screen "EQUIPO" 800x480
   GraphicView "Graphic view_1" at 621,5 size 174x31; Picture "LOGO CREMINOX (1)"
   Button "Button_17" at 13,1 size 45x40; TextOff 'Text'; PictureOff "Graphic_3"
      on Click: function_efd93a16()
   TextField "Text field_2" at 71,11 size 93x20; Text 'PARAMETROS'
   Button "Button_30" at 186,4 size 121x32; TextOff 'CONFIGURACION'
      on Click: ActivateScreen("MENU", 0)
   Button "Button_31" at 316,4 size 116x32; TextOff 'CERRAR SESION'
      on Click: function_f23ef4c9()
   Button "Button_12" at 445,5 size 102x32; TextOff 'RECETARIO'
      on Click: ActivateScreen("C RECETAS", 0)
      on Release: ResetBit("HMI RECETARIO")
      on Press: SetBit("HMI RECETARIO")
   TextField "Text field_27" at 301,189 size 50x20; Text 'VAPOR'
      Visibility <- "TIPO DE EQUIPO SELECCIONADO"
   TextField "Text field_28" at 307,208 size 37x20; Text 'VIVO'
      Visibility <- "TIPO DE EQUIPO SELECCIONADO"
   Switch "Switch_2" at 381,188 size 44x40; CaptionText 'Switch'; TextOff 'OFF'; TextOn 'ON'; PictureOn "Graphic_4"; PictureOff "Graphic_5"
      Visibility <- "TIPO DE EQUIPO SELECCIONADO"
      ProcessValue <- "ESTRUCTURAS Y ARREGLOS_HMI CARGA_VAPOR VIVO"
      on SwitchOn: SetBit("ESTRUCTURAS Y ARREGLOS_HMI CARGA_VAPOR VIVO")
      on SwitchOff: ResetBit("ESTRUCTURAS Y ARREGLOS_HMI CARGA_VAPOR VIVO")
   TextField "Text field_6" at 31,96 size 65x22; Text 'T. Agua:'
   IOField "I/O field_3" at 105,96 size 63x24; FormatPattern 99.9; Unit  °C
      ProcessValue <- "ESTRUCTURAS Y ARREGLOS_HMI CARGA_TEMPERATURAS_TEMPERATURA AGUA"
   TextField "Text field_8" at 200,96 size 86x22; Text 'T. Ingreso:'
   IOField "I/O field_4" at 299,96 size 63x24; FormatPattern 99.9; Unit  °C
      ProcessValue <- "ESTRUCTURAS Y ARREGLOS_HMI CARGA_TEMPERATURAS_TEMPERATURA INGRESO"
   TextField "Text field_9" at 391,96 size 63x22; Text 'T. Prod:'
   IOField "I/O field_5" at 468,96 size 63x24; FormatPattern 99.9; Unit  °C
      ProcessValue <- "ESTRUCTURAS Y ARREGLOS_HMI CARGA_TEMPERATURAS_TEMPERATURA PRODUCTO"
   TextField "Text field_7" at 559,96 size 112x22; Text 'Nivel de agua:'
   IOField "I/O field_13" at 686,96 size 69x25; FormatPattern 9999; Unit  mm
      ProcessValue <- "HMI NIVEL"
   TextField "Text field_3" at 28,132 size 153x22; Text 'PRE-OPERACIONAL'
   TextField "Text field_4" at 217,142 size 144x20; Text 'CANTIDAD DE TORRES'
   Button "Button_6" at 386,134 size 36x34; TextOff '-'
      on Press: SetBit("DISMINUIR CANT TORRES")
      on Release: ResetBit("DISMINUIR CANT TORRES")
      Visibility <- "VISUALIZACIONES HMI_LIM INF CANT TORRES"
   IOField "I/O field_6" at 435,133 size 41x35; FormatPattern 99
      ProcessValue <- "ESTRUCTURAS Y ARREGLOS_HMI CARGA_CANTIDAD DE TORRES"
   Button "Button_7" at 490,134 size 36x34; TextOff '+'
      on Press: SetBit("HMI AUMENTAR CANT TORRES")
      on Release: ResetBit("HMI AUMENTAR CANT TORRES")
      Visibility <- "VISUALIZACIONES HMI_LIM SUP CANT TORRES"
   TextField "Text field_23" at 35,210 size 52x20; Text 'TIEMPO'
      Visibility <- "ESTRUCTURAS Y ARREGLOS_HMI CARGA_TIPO DE CORTE"
   IOField "I/O field_1" at 134,202 size 81x32; FormatPattern 999; Unit  min
      ProcessValue <- "ESTRUCTURAS Y ARREGLOS_HMI CARGA_TIEMPO CORTE PC"
      Visibility <- "ESTRUCTURAS Y ARREGLOS_HMI CARGA_TIPO DE CORTE"
   TextField "Text field_5" at 12,178 size 128x20; Text 'POR TEMPERATURA'
   TextField "Text field_10" at 51,160 size 45x20; Text 'CORTE'
   Switch "Switch_1" at 153,159 size 47x38; CaptionText 'Switch'; TextOff 'OFF'; TextOn 'ON'; PictureOn "Graphic_4"; PictureOff "Graphic_5"
      ProcessValue <- "ESTRUCTURAS Y ARREGLOS_HMI CARGA_TIPO DE CORTE"
      on SwitchOn: SetBit("ESTRUCTURAS Y ARREGLOS_HMI CARGA_TIPO DE CORTE")
      on SwitchOff: ResetBit("ESTRUCTURAS Y ARREGLOS_HMI CARGA_TIPO DE CORTE")
   Button "Button_15" at 611,160 size 160x50; TextOff 'INICIAR PRE OP'
      on Release: ResetBit("INICIAR CICLO")
      on Press: SetBit("INICIAR CICLO")
      Visibility <- "ESTRUCTURAS Y ARREGLOS_HMI ESTADO_EN CICLO"
   TextField "Text field_11" at 14,210 size 98x20; Text 'TEMPERATURA'
      Visibility <- "ESTRUCTURAS Y ARREGLOS_HMI CARGA_TIPO DE CORTE"
   IOField "I/O field_15" at 135,202 size 81x32; FormatPattern 999; Unit  °C
      ProcessValue <- "ESTRUCTURAS Y ARREGLOS_HMI CARGA_TEMPERATURA CORTE PC"
      Visibility <- "ESTRUCTURAS Y ARREGLOS_HMI CARGA_TIPO DE CORTE"
   TextField "Text field_12" at 31,243 size 117x22; Text 'OPERACIONAL'
   TextField "Text field_13" at 31,270 size 110x20; Text 'RECETA ELEGIDA'
   TextField "Text field_15" at 31,308 size 129x20; Text 'NOMBRE DE RECETA'
   IOField "I/O field_8" at 196,303 size 221x27; FormatPattern ??????????????????????????
      ProcessValue <- "ESTRUCTURAS Y ARREGLOS_HMI CARGA_NOMBRE RECETA"
   Button "Button_8" at 207,260 size 36x34; TextOff '-'
      on Press: SetBit("HMI SEL ANT RECETA")
      on Release: ResetBit("HMI SEL ANT RECETA")
   IOField "I/O field_7" at 256,260 size 41x35; FormatPattern 99
      ProcessValue <- "HMI RECETA SELECCIONADA"
   Button "Button_9" at 311,261 size 36x34; TextOff '+'
      on Press: SetBit("HMI SEL SIG RECETA")
      on Release: ResetBit("HMI SEL SIG RECETA")
   Button "Button_10" at 367,261 size 129x33; TextOff 'VISUALIZAR'
      on Press: SetBit("HMI VISUALIZAR RECETA")
      on Release: ResetBit("HMI VISUALIZAR RECETA")
      on Click: ActivateScreen("C RECETAS", 0)
   Button "Button_16" at 608,262 size 161x50; TextOff 'INICIAR OPERACIONAL'
      on Release: ResetBit("HMI INICIAR CICLO OP")
      on Press: SetBit("HMI INICIAR CICLO OP")
      Visibility <- "ESTRUCTURAS Y ARREGLOS_HMI ESTADO_EN CICLO"
   TextField "Text field_18" at 30,352 size 114x20; Text 'ESTADO ACTUAL:'
   IOField "I/O field_9" at 153,347 size 251x27; FormatPattern ??????????????????????????????
      ProcessValue <- "ESTRUCTURAS Y ARREGLOS_HMI ESTADO_EQUIPO"
   TextField "Text field_20" at 429,351 size 199x20; Text 'TIEMPO TOTAL TRANSCURRIDO'
      Visibility <- "ESTRUCTURAS Y ARREGLOS_HMI ESTADO_EN CICLO"
   IOField "I/O field_10" at 639,346 size 81x32; FormatPattern 999; Unit  min
      ProcessValue <- "ESTRUCTURAS Y ARREGLOS_HMI ESTADO_TIEMPO TRANSCURRIDO"
      Visibility <- "ESTRUCTURAS Y ARREGLOS_HMI ESTADO_EN CICLO"
   TextField "Text field_21" at 29,392 size 98x20; Text 'PASO ACTUAL'
      Visibility <- "VISUALIZACIONES HMI_PASOS OP EN COCINAS"
   IOField "I/O field_11" at 143,383 size 41x35; FormatPattern 99
      Visibility <- "VISUALIZACIONES HMI_PASOS OP EN COCINAS"
      ProcessValue <- "ESTRUCTURAS Y ARREGLOS_HMI ESTADO_PASO ACTUAL"
   TextField "Text field_22" at 357,393 size 98x20; Text 'TIPO DE CORTE'
      Visibility <- "ESTRUCTURAS Y ARREGLOS_HMI ESTADO_EN CICLO"
   IOField "I/O field_12" at 469,389 size 194x27; FormatPattern ????????????????????
      Visibility <- "ESTRUCTURAS Y ARREGLOS_HMI ESTADO_EN CICLO"
      ProcessValue <- "ESTRUCTURAS Y ARREGLOS_HMI ESTADO_TIPO DE CORTE"
   Rectangle "Rectangle_2" at 1,126 size 798x354
      Visibility <- "ESTRUCTURAS Y ARREGLOS_HMI ESTADO_CICLO FINALIZADO"
   TextField "Text field_14" at 238,145 size 319x43; Text 'CICLO FINALIZADO'
      Visibility <- "ESTRUCTURAS Y ARREGLOS_HMI ESTADO_CICLO FINALIZADO"
   TextField "Text field_17" at 303,198 size 187x43; Text 'CON EXITO'
      Visibility <- "ESTRUCTURAS Y ARREGLOS_HMI ESTADO_CICLO FINALIZADO"
   GraphicView "Graphic view_2" at 348,251 size 98x92; Picture "Graphic_4"
      Visibility <- "ESTRUCTURAS Y ARREGLOS_HMI ESTADO_CICLO FINALIZADO"
   Button "Button_13" at 323,368 size 148x59; TextOff 'OK'
      Visibility <- "ESTRUCTURAS Y ARREGLOS_HMI ESTADO_CICLO FINALIZADO"
      on Press: SetBit("HMI OK FIN DE CICLO")
      on Release: ResetBit("HMI OK FIN DE CICLO")
   Rectangle "Rectangle_3" at 1,126 size 798x354
      Visibility <- "ESTRUCTURAS Y ARREGLOS_HMI ESTADO_CICLO CANCELADO"
   TextField "Text field_19" at 245,166 size 312x43; Text 'CICLO CANCELADO'
      Visibility <- "ESTRUCTURAS Y ARREGLOS_HMI ESTADO_CICLO CANCELADO"
   GraphicView "Graphic view_3" at 357,229 size 86x77; Picture "Graphic_5"
      Visibility <- "ESTRUCTURAS Y ARREGLOS_HMI ESTADO_CICLO CANCELADO"
   Button "Button_14" at 323,331 size 150x61; TextOff 'OK'
      Visibility <- "ESTRUCTURAS Y ARREGLOS_HMI ESTADO_CICLO CANCELADO"
      on Press: SetBit("HMI OK CANCELAR")
      on Release: ResetBit("HMI OK CANCELAR")
   Rectangle "Rectangle_4" at 1,126 size 798x113
      Visibility <- "ESTRUCTURAS Y ARREGLOS_HMI ESTADO_EN PO"
   Rectangle "Rectangle_5" at 1,238 size 798x100
      Visibility <- "ESTRUCTURAS Y ARREGLOS_HMI ESTADO_EN OP"
   Rectangle "Rectangle_6" at 2,128 size 796x112
      Visibility <- "ESTRUCTURAS Y ARREGLOS_HMI ESTADO_EN OP"
   Rectangle "Rectangle_8" at 599,139 size 185x183
      Visibility <- "ESTRUCTURAS Y ARREGLOS_HMI ESTADO_MANUAL ACTIVO"
   TextField "Text field_1" at 609,153 size 154x20; Text 'ACTUADORES ACTIVOS'
      Visibility <- "ESTRUCTURAS Y ARREGLOS_HMI ESTADO_MANUAL ACTIVO"
   TextField "Text field_24" at 623,175 size 127x20; Text 'EN FORMA MANUAL'
      Visibility <- "ESTRUCTURAS Y ARREGLOS_HMI ESTADO_MANUAL ACTIVO"
   Button "Button_11" at 642,261 size 98x38; TextOff 'RESET'
      Visibility <- "ESTRUCTURAS Y ARREGLOS_HMI ESTADO_MANUAL ACTIVO"
      on Press: SetBit("HMI RESET ACTUADORES MANUAL")
      on Release: ResetBit("HMI RESET ACTUADORES MANUAL")
   TextField "Text field_25" at 623,197 size 126x20; Text 'PULSE RESET PARA'
      Visibility <- "ESTRUCTURAS Y ARREGLOS_HMI ESTADO_MANUAL ACTIVO"
   TextField "Text field_26" at 629,220 size 115x20; Text 'DESACTIVARLOS'
      Visibility <- "ESTRUCTURAS Y ARREGLOS_HMI ESTADO_MANUAL ACTIVO"
   Button "Button_3" at 25,429 size 97x43; TextOff 'CANCELAR'
      on Release: ResetBit("HMI CANCELAR")
      on Press: SetBit("HMI CANCELAR")
      Visibility <- "ESTRUCTURAS Y ARREGLOS_HMI ESTADO_PULSADOR CANCELAR"
   Button "Button_4" at 136,430 size 97x43; TextOff 'CONTINUAR'
      on Release: ResetBit("HMI CONTINUAR")
      on Press: SetBit("HMI CONTINUAR")
      Visibility <- "ESTRUCTURAS Y ARREGLOS_HMI ESTADO_PULSADOR CONTINUAR"
   Button "Button_5" at 249,430 size 97x43; TextOff 'PAUSAR'
      on Release: ResetBit("HMI PAUSA")
      on Press: SetBit("HMI PAUSA")
      Visibility <- "ESTRUCTURAS Y ARREGLOS_HMI ESTADO_PULSADOR PAUSA"
   IOField "I/O field_16" at 166,49 size 215x35; FormatPattern ??????????????????????????
      ProcessValue <- "ESTRUCTURAS Y ARREGLOS_HMI NOMBRE EQUIPO"
   Button "Button_19" at 400,49 size 39x35; TextOff 'Text'; PictureOff "Graphic_1"
      on Release: ResetBit("HMI DISMINUIR EQUIPO")
      on Press: SetBit("HMI DISMINUIR EQUIPO")
      Visibility <- "VISUALIZACIONES HMI_LIM INF EQUIPO SEL"
   IOField "I/O field_2" at 464,49 size 42x35; FormatPattern 99
      ProcessValue <- "EQUIPO SELECCIONADO"
   Button "Button_18" at 531,49 size 40x35; TextOff 'Text'; PictureOff "Graphic_2"
      on Release: ResetBit("HMI AUMENTAR EQUIPO")
      on Press: SetBit("HMI AUMENTAR EQUIPO")
      Visibility <- "VISUALIZACIONES HMI_LIM SUP EQUIPO SEL"
   Button "Button_1" at 567,434 size 183x37; TextOff 'GRAFICO TEMPERATURAS'
      on Click: ActivateScreen("GRAFICOS", 0)
   Button "Button_2" at 204,384 size 109x35; TextOff 'SALTAR PASO'
      on Press: SetBit("HMI SALTAR PASO")
      on Release: ResetBit("HMI SALTAR PASO")
      Visibility <- "VISUALIZACIONES HMI_PASOS OP EN COCINAS"

screen "C GENERALES" 800x480
   TextField "Text field_7" at 439,158 size 246x29; Text 'Histeresis temperatura'
   IOField "I/O field_4" at 706,153 size 74x40; FormatPattern 999; Unit  °C
      ProcessValue <- "ESTRUCTURAS Y ARREGLOS_HMI CONFIGURACION_HISTERESIS"
   TextField "Text field_8" at 28,338 size 228x29; Text 'Tiempo Maximo Ciclo'
   IOField "I/O field_5" at 326,333 size 74x40; FormatPattern 999; Unit  min
      ProcessValue <- "ESTRUCTURAS Y ARREGLOS_HMI CONFIGURACION_TIEMPO MAXIMO CICLO"
   IOField "I/O field_3" at 326,242 size 74x40; FormatPattern 9999; Unit  mm
      ProcessValue <- "ESTRUCTURAS Y ARREGLOS_HMI CONFIGURACION_NIVEL CRITICO OP"
   TextField "Text field_9" at 26,158 size 281x29; Text 'Nivel Critico Pre-operativo'
   IOField "I/O field_10" at 326,153 size 74x40; FormatPattern 9999; Unit  mm
      ProcessValue <- "ESTRUCTURAS Y ARREGLOS_HMI CONFIGURACION_NIVEL CRITICO"
   GraphicView "Graphic view_1" at 621,4 size 174x31; Picture "LOGO CREMINOX (1)"
   TextField "Text field_1" at 213,106 size 14x20; Text 'Text'
   Button "Button_1" at 734,430 size 40x35; TextOff 'Text'; PictureOff "Graphic_2"
      on Click: ActivateScreen("C NIVELES PO Y OP", 0)
   Button "Button_4" at 28,430 size 39x35; TextOff 'Text'; PictureOff "Graphic_1"
      on Click: ActivateScreen("C TEMPERATURAS", 0)
   Button "Button_6" at 17,2 size 40x38; TextOff 'Text'; PictureOff "Home"
      on Click: ActivateScreen("PRINCIPAL", 0)
   TextField "Text field_2" at 145,12 size 196x20; Text 'CONFIGURACIONES GENERALES'
   TextField "Text field_3" at 76,439 size 156x18; Text 'A CONF. TEMPERATURAS'
   TextField "Text field_4" at 615,439 size 107x18; Text 'A CONF. NIVELES'
   Button "Button_17" at 83,1 size 45x40; TextOff 'Text'; PictureOff "Graphic_3"
      on Click: ActivateScreen("MENU", 0)
   TextField "Text field_5" at 28,247 size 237x29; Text 'Nivel Critico operativo'
   IOField "I/O field_16" at 166,55 size 215x35; FormatPattern ??????????????????????????
      ProcessValue <- "ESTRUCTURAS Y ARREGLOS_HMI NOMBRE EQUIPO"
   Button "Button_19" at 400,55 size 39x35; TextOff 'Text'; PictureOff "Graphic_1"
      on Release: ResetBit("HMI DISMINUIR EQUIPO")
      on Press: SetBit("HMI DISMINUIR EQUIPO")
      Visibility <- "VISUALIZACIONES HMI_LIM INF EQUIPO SEL"
   IOField "I/O field_1" at 464,55 size 42x35; FormatPattern 99
      ProcessValue <- "EQUIPO SELECCIONADO"
   Button "Button_18" at 531,55 size 40x35; TextOff 'Text'; PictureOff "Graphic_2"
      on Release: ResetBit("HMI AUMENTAR EQUIPO")
      on Press: SetBit("HMI AUMENTAR EQUIPO")
      Visibility <- "VISUALIZACIONES HMI_LIM SUP EQUIPO SEL"

screen "C RECETAS" 800x480
   TextField "Text field_18" at 328,196 size 142x20; Text 'TEMPERATURA CORTE'
      Visibility <- "VISUALIZACIONES HMI_TIPO DE CORTE PASO 1"
   IOField "I/O field_9" at 495,193 size 73x27; FormatPattern 999; Unit  °C
      ProcessValue <- "ESTRUCTURAS Y ARREGLOS_HMI EDICION RECETAS_TEMP PRODUCTO{1}"
      Visibility <- "VISUALIZACIONES HMI_TIPO DE CORTE PASO 1"
   TextField "Text field_19" at 328,240 size 142x20; Text 'TEMPERATURA CORTE'
      Visibility <- "VISUALIZACIONES HMI_TIPO DE CORTE PASO 2"
   IOField "I/O field_10" at 495,236 size 74x27; FormatPattern 999; Unit  °C
      ProcessValue <- "ESTRUCTURAS Y ARREGLOS_HMI EDICION RECETAS_TEMP PRODUCTO{2}"
      Visibility <- "VISUALIZACIONES HMI_TIPO DE CORTE PASO 2"
   TextField "Text field_20" at 328,285 size 142x20; Text 'TEMPERATURA CORTE'
      Visibility <- "VISUALIZACIONES HMI_TIPO DE CORTE PASO 3"
   IOField "I/O field_11" at 495,281 size 73x27; FormatPattern 999; Unit  °C
      ProcessValue <- "ESTRUCTURAS Y ARREGLOS_HMI EDICION RECETAS_TEMP PRODUCTO{3}"
      Visibility <- "VISUALIZACIONES HMI_TIPO DE CORTE PASO 3"
   TextField "Text field_21" at 328,332 size 142x20; Text 'TEMPERATURA CORTE'
      Visibility <- "VISUALIZACIONES HMI_TIPO DE CORTE PASO 4"
   IOField "I/O field_12" at 495,328 size 73x27; FormatPattern 999; Unit  °C
      ProcessValue <- "ESTRUCTURAS Y ARREGLOS_HMI EDICION RECETAS_TEMP PRODUCTO{4}"
      Visibility <- "VISUALIZACIONES HMI_TIPO DE CORTE PASO 4"
   TextField "Text field_26" at 327,399 size 142x20; Text 'TEMPERATURA CORTE'
      Visibility <- "VISUALIZACIONES HMI_CORTE TEMP ENFRIADOR"
   IOField "I/O field_17" at 496,396 size 73x27; FormatPattern 999; Unit  °C
      ProcessValue <- "ESTRUCTURAS Y ARREGLOS_HMI EDICION RECETAS_TEMP CORTE ENFRIADO"
      Visibility <- "VISUALIZACIONES HMI_CORTE TEMP ENFRIADOR"
   GraphicView "Graphic view_1" at 620,6 size 174x31; Picture "LOGO CREMINOX (1)"
   TextField "Text field_3" at 20,113 size 129x20; Text 'NOMBRE DE RECETA'
   IOField "I/O field_2" at 167,108 size 220x32; FormatPattern ?????????????????????????
      ProcessValue <- "ESTRUCTURAS Y ARREGLOS_HMI EDICION RECETAS_NOMBRE"
   TextField "Text field_4" at 673,66 size 48x20; Text 'PASOS'
   Button "Button_6" at 630,103 size 33x30; TextOff '-'
      on Press: SetBit("HMI RESTAR PASO")
      on Release: ResetBit("HMI RESTAR PASO")
      Visibility <- "VISUALIZACIONES HMI_ANTERIOR PASO"
   Button "Button_7" at 732,102 size 34x31; TextOff '+'
      on Press: SetBit("HMI SUMAR PASO")
      on Release: ResetBit("HMI SUMAR PASO")
      Visibility <- "VISUALIZACIONES HMI_SIGUIENTE PASO"
   IOField "I/O field_6" at 677,101 size 41x32; FormatPattern 99
      ProcessValue <- "ESTRUCTURAS Y ARREGLOS_HMI EDICION RECETAS_PASOS"
   TextField "Text field_5" at 31,196 size 52x20; Text 'PASO 1'
      Visibility <- "VISUALIZACIONES HMI_1 PASO RECETA"
   TextField "Text field_6" at 31,240 size 52x20; Text 'PASO 2'
      Visibility <- "VISUALIZACIONES HMI_2 PASOS RECETA"
   TextField "Text field_7" at 31,285 size 52x20; Text 'PASO 3'
      Visibility <- "VISUALIZACIONES HMI_3 PASOS RECETA"
   TextField "Text field_8" at 31,330 size 52x20; Text 'PASO 4'
      Visibility <- "VISUALIZACIONES HMI_4 PASOS RECETA"
   TextField "Text field_22" at 672,141 size 45x20; Text 'CORTE'
   TextField "Text field_23" at 31,151 size 61x20; Text 'COCINAS'
   TextField "Text field_24" at 22,362 size 92x20; Text 'ENFRIADORES'
   Button "Button_18" at 526,56 size 40x35; TextOff 'Text'; PictureOff "Graphic_2"
      on Release: ResetBit("HMI RECETA SIGUIENTE")
      on Press: SetBit("HMI RECETA SIGUIENTE")
      Visibility <- "VISUALIZACIONES HMI_SIGUIENTE RECETA"
   Button "Button_19" at 405,55 size 39x35; TextOff 'Text'; PictureOff "Graphic_1"
      on Release: ResetBit("HMI RECETA ANTERIOR")
      on Press: SetBit("HMI RECETA ANTERIOR")
      Visibility <- "VISUALIZACIONES HMI_ANTERIOR RECETA"
   Button "Button_1" at 740,437 size 40x35; TextOff 'Text'; PictureOff "Graphic_2"
      on Click: ActivateScreen("C REGLA", 0)
      Visibility <- "VISUALIZACIONES HMI_BLOQUEO EDICION RECETAS"
   Button "Button_2" at 20,437 size 39x35; TextOff 'Text'; PictureOff "Graphic_1"
      on Click: ActivateScreen("C NIVELES PO Y OP", 0)
      Visibility <- "VISUALIZACIONES HMI_BLOQUEO EDICION RECETAS"
   TextField "Text field_10" at 79,11 size 61x20; Text 'RECETAS'
   TextField "Text field_27" at 72,444 size 112x18; Text 'A CONF. RECETAS'
      Visibility <- "VISUALIZACIONES HMI_BLOQUEO EDICION RECETAS"
   TextField "Text field_28" at 628,446 size 97x18; Text 'A CONF. REGLA'
      Visibility <- "VISUALIZACIONES HMI_BLOQUEO EDICION RECETAS"
   TextField "Text field_29" at 631,159 size 128x20; Text 'POR TEMPERATURA'
   Switch "Switch_1" at 676,187 size 43x38; CaptionText 'Switch'; TextOff 'OFF'; TextOn 'ON'; PictureOn "Graphic_4"; PictureOff "Graphic_5"
      ProcessValue <- "ESTRUCTURAS Y ARREGLOS_HMI EDICION RECETAS_TIPO CORTE{1}"
      Visibility <- "VISUALIZACIONES HMI_1 PASO RECETA"
   Switch "Switch_2" at 676,229 size 43x38; CaptionText 'Switch'; TextOff 'OFF'; TextOn 'ON'; PictureOff "Graphic_5"; PictureOn "Graphic_4"
      ProcessValue <- "ESTRUCTURAS Y ARREGLOS_HMI EDICION RECETAS_TIPO CORTE{2}"
      Visibility <- "VISUALIZACIONES HMI_2 PASOS RECETA"
   Switch "Switch_3" at 676,275 size 43x38; CaptionText 'Switch'; TextOff 'OFF'; TextOn 'ON'; PictureOff "Graphic_5"; PictureOn "Graphic_4"
      ProcessValue <- "ESTRUCTURAS Y ARREGLOS_HMI EDICION RECETAS_TIPO CORTE{3}"
      Visibility <- "VISUALIZACIONES HMI_3 PASOS RECETA"
   Switch "Switch_4" at 676,319 size 43x38; CaptionText 'Switch'; TextOff 'OFF'; TextOn 'ON'; PictureOff "Graphic_5"; PictureOn "Graphic_4"
      ProcessValue <- "ESTRUCTURAS Y ARREGLOS_HMI EDICION RECETAS_TIPO CORTE{4}"
      Visibility <- "VISUALIZACIONES HMI_4 PASOS RECETA"
   Switch "Switch_5" at 676,389 size 43x38; CaptionText 'Switch'; TextOff 'OFF'; TextOn 'ON'; PictureOff "Graphic_5"; PictureOn "Graphic_4"
      ProcessValue <- "ESTRUCTURAS Y ARREGLOS_HMI EDICION RECETAS_TIPO CORTE ENFRIADO"
   Button "Button_17" at 13,0 size 45x40; TextOff 'Text'; PictureOff "Graphic_3"
      on Click: function_efd93a16()
      on Press: SetBit("HMI VOLVER")
      on Release: ResetBit("HMI VOLVER")
   TextField "Text field_14" at 337,197 size 116x20; Text 'TIEMPO DE CORTE'
      Visibility <- "VISUALIZACIONES HMI_CORTE TIEMPO PASO 1"
   IOField "I/O field_14" at 495,194 size 74x27; FormatPattern 999; Unit  min
      ProcessValue <- "ESTRUCTURAS Y ARREGLOS_HMI EDICION RECETAS_TIEMPO CORTE{1}"
      Visibility <- "VISUALIZACIONES HMI_CORTE TIEMPO PASO 1"
   TextField "Text field_15" at 337,239 size 116x20; Text 'TIEMPO DE CORTE'
      Visibility <- "VISUALIZACIONES HMI_CORTE TIEMPO PASO 2"
   IOField "I/O field_3" at 496,236 size 74x27; FormatPattern 999; Unit  min
      ProcessValue <- "ESTRUCTURAS Y ARREGLOS_HMI EDICION RECETAS_TIEMPO CORTE{2}"
      Visibility <- "VISUALIZACIONES HMI_CORTE TIEMPO PASO 2"
   TextField "Text field_16" at 338,282 size 116x20; Text 'TIEMPO DE CORTE'
      Visibility <- "VISUALIZACIONES HMI_CORTE TIEMPO PASO 3"
   IOField "I/O field_15" at 495,279 size 74x27; FormatPattern 999; Unit  min
      ProcessValue <- "ESTRUCTURAS Y ARREGLOS_HMI EDICION RECETAS_TIEMPO CORTE{3}"
      Visibility <- "VISUALIZACIONES HMI_CORTE TIEMPO PASO 3"
   TextField "Text field_17" at 337,325 size 116x20; Text 'TIEMPO DE CORTE'
      Visibility <- "VISUALIZACIONES HMI_CORTE TIEMPO PASO 4"
   IOField "I/O field_16" at 495,322 size 74x27; FormatPattern 999; Unit  min
      ProcessValue <- "ESTRUCTURAS Y ARREGLOS_HMI EDICION RECETAS_TIEMPO CORTE{4}"
      Visibility <- "VISUALIZACIONES HMI_CORTE TIEMPO PASO 4"
   TextField "Text field_1" at 336,404 size 116x20; Text 'TIEMPO DE CORTE'
      Visibility <- "VISUALIZACIONES HMI_CORTE TIEMPO ENFRIADOR"
   IOField "I/O field_13" at 494,398 size 74x27; FormatPattern 999; Unit  min
      ProcessValue <- "ESTRUCTURAS Y ARREGLOS_HMI EDICION RECETAS_TIEMPO CORTE ENFRIADO"
      Visibility <- "VISUALIZACIONES HMI_CORTE TIEMPO ENFRIADOR"
   TextField "Text field_2" at 237,57 size 129x33; Text 'NUMERO DE RECETA'
   IOField "I/O field_1" at 464,56 size 42x35; FormatPattern 99
      ProcessValue <- "HMI NUMERO RECETA"
   TextField "Text field_9" at 122,196 size 82x20; Text 'TEMP. AGUA'
      Visibility <- "VISUALIZACIONES HMI_1 PASO RECETA"
   IOField "I/O field_4" at 239,193 size 68x27; FormatPattern 999; Unit  °C
      ProcessValue <- "ESTRUCTURAS Y ARREGLOS_HMI EDICION RECETAS_TEMP AGUA{1}"
      Visibility <- "VISUALIZACIONES HMI_1 PASO RECETA"
   TextField "Text field_11" at 122,240 size 82x20; Text 'TEMP. AGUA'
      Visibility <- "VISUALIZACIONES HMI_2 PASOS RECETA"
   IOField "I/O field_5" at 238,236 size 68x27; FormatPattern 999; Unit  °C
      ProcessValue <- "ESTRUCTURAS Y ARREGLOS_HMI EDICION RECETAS_TEMP AGUA{2}"
      Visibility <- "VISUALIZACIONES HMI_2 PASOS RECETA"
   TextField "Text field_12" at 122,285 size 82x20; Text 'TEMP. AGUA'
      Visibility <- "VISUALIZACIONES HMI_3 PASOS RECETA"
   IOField "I/O field_7" at 238,281 size 68x27; FormatPattern 999; Unit  °C
      ProcessValue <- "ESTRUCTURAS Y ARREGLOS_HMI EDICION RECETAS_TEMP AGUA{3}"
      Visibility <- "VISUALIZACIONES HMI_3 PASOS RECETA"
   TextField "Text field_13" at 122,331 size 82x20; Text 'TEMP. AGUA'
      Visibility <- "VISUALIZACIONES HMI_4 PASOS RECETA"
   IOField "I/O field_8" at 238,329 size 68x27; FormatPattern 999; Unit  °C
      ProcessValue <- "ESTRUCTURAS Y ARREGLOS_HMI EDICION RECETAS_TEMP AGUA{4}"
      Visibility <- "VISUALIZACIONES HMI_4 PASOS RECETA"
   Rectangle "Rectangle_2" at 5,95 size 789x382
      Visibility <- "VISUALIZACIONES HMI_BLOQUEO EDICION RECETAS"

screen "C NIVELES PO Y OP" 800x480
   GraphicView "Graphic view_1" at 621,4 size 174x31; Picture "LOGO CREMINOX (1)"
   TextField "Text field_1" at 568,205 size 99x27; Text 'Operativo'
   TextField "Text field_6" at 117,205 size 136x27; Text 'Pre Operativo'
   TextField "Text field_7" at 119,205 size 18x27; Text 'Text'
   IOField "I/O field_1" at 592,121 size 72x34; FormatPattern 9999; Unit  mm
      ProcessValue <- "ESTRUCTURAS Y ARREGLOS_HMI CONFIGURACION_VENTANA"
   TextField "Text field_8" at 91,257 size 74x27; Text '1 Torre'
   TextField "Text field_13" at 477,124 size 83x27; Text 'Ventana'
   IOField "I/O field_9" at 193,254 size 74x34; FormatPattern 9999; Unit  mm
      ProcessValue <- "ESTRUCTURAS Y ARREGLOS_HMI CONFIGURACION_NIVEL PO{1}"
   IOField "I/O field_21" at 242,121 size 72x34; FormatPattern 9999; Unit  mm
      ProcessValue <- "HMI NIVEL"
   IOField "I/O field_25" at 576,251 size 75x34; FormatPattern 9999; Unit  mm
      ProcessValue <- "ESTRUCTURAS Y ARREGLOS_HMI CONFIGURACION_NIVEL OP"
   TextField "Text field_12" at 83,124 size 120x27; Text 'Nivel Actual'
   Button "Button_1" at 734,430 size 40x35; TextOff 'Text'; PictureOff "Graphic_2"
      on Click: ActivateScreen("C RECETAS", 0)
   Button "Button_2" at 28,430 size 39x35; TextOff 'Text'; PictureOff "Graphic_1"
      on Click: ActivateScreen("C GENERALES", 0)
   Button "Button_6" at 17,2 size 40x38; TextOff 'Text'; PictureOff "Home"
      on Click: ActivateScreen("PRINCIPAL", 0)
   TextField "Text field_2" at 142,12 size 56x20; Text 'NIVELES'
   TextField "Text field_3" at 76,439 size 127x18; Text 'A CONF. GENERALES'
   TextField "Text field_4" at 603,439 size 112x18; Text 'A CONF. RECETAS'
   Button "Button_17" at 81,0 size 45x40; TextOff 'Text'; PictureOff "Graphic_3"
      on Click: function_efd93a16()
   IOField "I/O field_16" at 166,54 size 215x35; FormatPattern ??????????????????????????
      ProcessValue <- "ESTRUCTURAS Y ARREGLOS_HMI NOMBRE EQUIPO"
   Button "Button_19" at 400,54 size 39x35; TextOff 'Text'; PictureOff "Graphic_1"
      on Release: ResetBit("HMI DISMINUIR EQUIPO")
      on Press: SetBit("HMI DISMINUIR EQUIPO")
      Visibility <- "VISUALIZACIONES HMI_LIM INF EQUIPO SEL"
   IOField "I/O field_2" at 464,54 size 42x35; FormatPattern 99
      ProcessValue <- "EQUIPO SELECCIONADO"
   Button "Button_18" at 531,54 size 40x35; TextOff 'Text'; PictureOff "Graphic_2"
      on Release: ResetBit("HMI AUMENTAR EQUIPO")
      on Press: SetBit("HMI AUMENTAR EQUIPO")
      Visibility <- "VISUALIZACIONES HMI_LIM SUP EQUIPO SEL"

screen "C TEMPERATURAS" 800x480
   IOField "I/O field_1" at 161,153 size 69x32; FormatPattern 99.9; Unit  °C
      ProcessValue <- "ESTRUCTURAS Y ARREGLOS_HMI CARGA_TEMPERATURAS_TEMPERATURA AGUA SC"
   TextField "Text field_1" at 30,158 size 97x22; Text 'TEMP. AGUA'
   TextField "Text field_4" at 300,158 size 63x22; Text 'OFFSET'
   TextField "Text field_5" at 531,158 size 97x22; Text 'CORREGIDA'
   IOField "I/O field_3" at 658,153 size 69x32; FormatPattern 99.9; Unit  °C
      ProcessValue <- "ESTRUCTURAS Y ARREGLOS_HMI CARGA_TEMPERATURAS_TEMPERATURA AGUA"
   IOField "I/O field_4" at 161,252 size 69x32; FormatPattern 99.9; Unit  °C
      ProcessValue <- "ESTRUCTURAS Y ARREGLOS_HMI CARGA_TEMPERATURAS_TEMPERATURA INGRESO SC"
   TextField "Text field_2" at 15,257 size 127x22; Text 'TEMP. INGRESO'
   TextField "Text field_3" at 300,257 size 63x22; Text 'OFFSET'
   TextField "Text field_6" at 531,256 size 97x22; Text 'CORREGIDA'
   IOField "I/O field_5" at 383,252 size 69x32; FormatPattern 99.9; Unit  °C
      ProcessValue <- "ESTRUCTURAS Y ARREGLOS_CORRECCIONES HMI_TEMPERATURA INGRESO SC"
   IOField "I/O field_6" at 658,252 size 69x32; FormatPattern 99.9; Unit  °C
      ProcessValue <- "ESTRUCTURAS Y ARREGLOS_HMI CARGA_TEMPERATURAS_TEMPERATURA INGRESO"
   IOField "I/O field_7" at 161,349 size 69x32; FormatPattern 99.9; Unit  °C
      ProcessValue <- "ESTRUCTURAS Y ARREGLOS_HMI CARGA_TEMPERATURAS_TEMPERATURA PRODUCTO SC"
   TextField "Text field_7" at 8,356 size 141x22; Text 'TEMP. PRODUCTO'
   TextField "Text field_8" at 300,354 size 63x22; Text 'OFFSET'
   TextField "Text field_9" at 531,354 size 97x22; Text 'CORREGIDA'
   IOField "I/O field_8" at 385,349 size 69x32; FormatPattern 99.9; Unit  °C
      ProcessValue <- "ESTRUCTURAS Y ARREGLOS_CORRECCIONES HMI_TEMPERATURA PRODUCTO SC"
   IOField "I/O field_9" at 658,349 size 69x32; FormatPattern 99.9; Unit  °C
      ProcessValue <- "ESTRUCTURAS Y ARREGLOS_HMI CARGA_TEMPERATURAS_TEMPERATURA PRODUCTO"
   GraphicView "Graphic view_1" at 620,5 size 174x31; Picture "LOGO CREMINOX (1)"
   TextField "Text field_10" at 248,158 size 34x23; Text '+/-'
   TextField "Text field_11" at 481,158 size 18x23; Text '='
   TextField "Text field_12" at 248,257 size 34x23; Text '+/-'
   TextField "Text field_13" at 481,257 size 18x23; Text '='
   TextField "Text field_14" at 248,354 size 34x23; Text '+/-'
   TextField "Text field_15" at 481,354 size 18x23; Text '='
   IOField "I/O field_2" at 386,153 size 69x32; FormatPattern 99.9; Unit  °C
      ProcessValue <- "ESTRUCTURAS Y ARREGLOS_CORRECCIONES HMI_TEMPERATURA AGUA SC"
   Button "Button_3" at 734,430 size 40x35; TextOff 'Text'; PictureOff "Graphic_2"
      on Click: ActivateScreen("C GENERALES", 0)
   Button "Button_4" at 28,430 size 39x35; TextOff 'Text'; PictureOff "Graphic_1"
      on Click: ActivateScreen("C REGLA", 0)
   Button "Button_6" at 17,2 size 40x38; TextOff 'Text'; PictureOff "Home"
      on Click: ActivateScreen("PRINCIPAL", 0)
   TextField "Text field_16" at 152,12 size 295x20; Text 'CORRECCION EN MEDICION DE TEMPERATURAS'
   TextField "Text field_28" at 82,439 size 156x18; Text 'A CONF. TEMPERATURAS'
   TextField "Text field_17" at 595,439 size 127x18; Text 'A CONF. GENERALES'
   Button "Button_17" at 82,1 size 45x40; TextOff 'Text'; PictureOff "Graphic_3"
      on Click: function_efd93a16()
   IOField "I/O field_16" at 166,54 size 215x35; FormatPattern ??????????????????????????
      ProcessValue <- "ESTRUCTURAS Y ARREGLOS_HMI NOMBRE EQUIPO"
   Button "Button_19" at 400,54 size 39x35; TextOff 'Text'; PictureOff "Graphic_1"
      on Release: ResetBit("HMI DISMINUIR EQUIPO")
      on Press: SetBit("HMI DISMINUIR EQUIPO")
      Visibility <- "VISUALIZACIONES HMI_LIM INF EQUIPO SEL"
   IOField "I/O field_10" at 464,54 size 42x35; FormatPattern 99
      ProcessValue <- "EQUIPO SELECCIONADO"
   Button "Button_18" at 531,54 size 40x35; TextOff 'Text'; PictureOff "Graphic_2"
      on Release: ResetBit("HMI AUMENTAR EQUIPO")
      on Press: SetBit("HMI AUMENTAR EQUIPO")
      Visibility <- "VISUALIZACIONES HMI_LIM SUP EQUIPO SEL"

screen "C REGLA" 800x480
   Button "Button_1" at 443,158 size 97x47; TextOff 'OK'
      on Press: SetBit("CALIBRACION SN MAXIMO")
      on Release: ResetBit("CALIBRACION SN MAXIMO")
   Button "Button_2" at 441,253 size 97x47; TextOff 'OK'
      on Press: SetBit("CALIBRACION SN MINIMO")
      on Release: ResetBit("CALIBRACION SN MINIMO")
   TextField "Text field_1" at 258,171 size 129x23; Text 'NIVEL MAXIMO'
   TextField "Text field_2" at 258,268 size 129x23; Text 'NIVEL MINIMO'
   TextField "Text field_3" at 258,366 size 129x23; Text 'NIVEL ACTUAL'
   IOField "I/O field_1" at 441,355 size 98x45; FormatPattern 99999; Unit  mm
      ProcessValue <- "HMI NIVEL"
   GraphicView "Graphic view_1" at 620,5 size 174x31; Picture "LOGO CREMINOX (1)"
   Button "Button_3" at 734,430 size 40x35; TextOff 'Text'; PictureOff "Graphic_2"
      on Click: ActivateScreen("C TEMPERATURAS", 0)
   Button "Button_4" at 28,430 size 39x35; TextOff 'Text'; PictureOff "Graphic_1"
      on Click: ActivateScreen("C RECETAS", 0)
   Button "Button_6" at 17,2 size 40x38; TextOff 'Text'; PictureOff "Home"
      on Click: ActivateScreen("PRINCIPAL", 0)
   TextField "Text field_10" at 151,11 size 151x20; Text 'CONFIGURACION REGLA'
   TextField "Text field_28" at 82,439 size 97x18; Text 'A CONF. REGLA'
   TextField "Text field_4" at 559,440 size 156x18; Text 'A CONF. TEMPERATURAS'
   Button "Button_17" at 89,0 size 45x40; TextOff 'Text'; PictureOff "Graphic_3"
      on Click: function_efd93a16()
   IOField "I/O field_16" at 166,59 size 215x35; FormatPattern ??????????????????????????
      ProcessValue <- "ESTRUCTURAS Y ARREGLOS_HMI NOMBRE EQUIPO"
   Button "Button_19" at 400,59 size 39x35; TextOff 'Text'; PictureOff "Graphic_1"
      on Release: ResetBit("HMI DISMINUIR EQUIPO")
      on Press: SetBit("HMI DISMINUIR EQUIPO")
      Visibility <- "VISUALIZACIONES HMI_LIM INF EQUIPO SEL"
   IOField "I/O field_2" at 464,59 size 42x35; FormatPattern 99
      ProcessValue <- "EQUIPO SELECCIONADO"
   Button "Button_18" at 531,59 size 40x35; TextOff 'Text'; PictureOff "Graphic_2"
      on Release: ResetBit("HMI AUMENTAR EQUIPO")
      on Press: SetBit("HMI AUMENTAR EQUIPO")
      Visibility <- "VISUALIZACIONES HMI_LIM SUP EQUIPO SEL"

screen "MENU" 800x480
   GraphicView "Graphic view_1" at 621,4 size 174x31; Picture "LOGO CREMINOX (1)"
   Button "Button_1" at 339,75 size 121x53; TextOff 'GENERALES'
      on Click: ActivateScreen("C GENERALES", 0)
   Button "Button_2" at 321,228 size 158x53; TextOff 'EDICION DE RECETAS'
      on Click: ActivateScreen("C RECETAS", 0)
   Button "Button_3" at 311,305 size 177x53; TextOff 'CALIBRACION DE REGLA'
      on Click: ActivateScreen("C REGLA", 0)
   Button "Button_4" at 282,382 size 235x53; TextOff 'CALIBRACION DE TEMPERATURAS'
      on Click: ActivateScreen("C TEMPERATURAS", 0)
   Button "Button_5" at 339,151 size 121x53; TextOff 'NIVELES'
      on Click: ActivateScreen("C NIVELES PO Y OP", 0)
   TextField "Text field_10" at 73,12 size 106x20; Text 'CONFIGURACION'
   Button "Button_17" at 13,2 size 45x40; TextOff 'Text'; PictureOff "Graphic_3"
      on Click: function_efd93a16()
   Button "Button_11" at 213,4 size 96x32; TextOff 'MANUAL'
      on Click: ActivateScreen("MANUAL", 0)
   Button "Button_26" at 333,5 size 116x32; TextOff 'CERRAR SESION'
      on Click: function_f23ef4c9()

screen "GRAFICOS" 800x480
   GraphicView "Graphic view_1" at 621,5 size 174x31; Picture "LOGO CREMINOX (1)"
   Button "Button_17" at 13,2 size 45x40; TextOff 'Text'; PictureOff "Graphic_3"
      on Click: function_efd93a16()
   TextField "Text field_10" at 88,12 size 245x20; Text 'GRAFICOS TEMPERATURAS VS TIEMPO'
   IOField "I/O field_16" at 166,47 size 215x35; FormatPattern ??????????????????????????
      ProcessValue <- "ESTRUCTURAS Y ARREGLOS_HMI NOMBRE EQUIPO"
   Button "Button_19" at 400,47 size 39x35; TextOff 'Text'; PictureOff "Graphic_1"
      on Release: ResetBit("HMI DISMINUIR EQUIPO")
      on Press: SetBit("HMI DISMINUIR EQUIPO")
      Visibility <- "VISUALIZACIONES HMI_LIM INF EQUIPO SEL"
   IOField "I/O field_2" at 464,47 size 42x35; FormatPattern 99
      ProcessValue <- "EQUIPO SELECCIONADO"
   Button "Button_18" at 531,47 size 40x35; TextOff 'Text'; PictureOff "Graphic_2"
      on Release: ResetBit("HMI AUMENTAR EQUIPO")
      on Press: SetBit("HMI AUMENTAR EQUIPO")
      Visibility <- "VISUALIZACIONES HMI_LIM SUP EQUIPO SEL"
   TrendView "Trend view_1" at 10,90 size 780x384
      Visibility <- "VISUALIZACIONES HMI_GRAFICOS"
   TrendView "Trend view_2" at 10,90 size 780x384
      Visibility <- "VISUALIZACIONES HMI_GRAFICOS"
*)